// Mitsubishi GX Works2 project: 단속동작   PLC: Q02/Q02H

PROGRAM MAIN
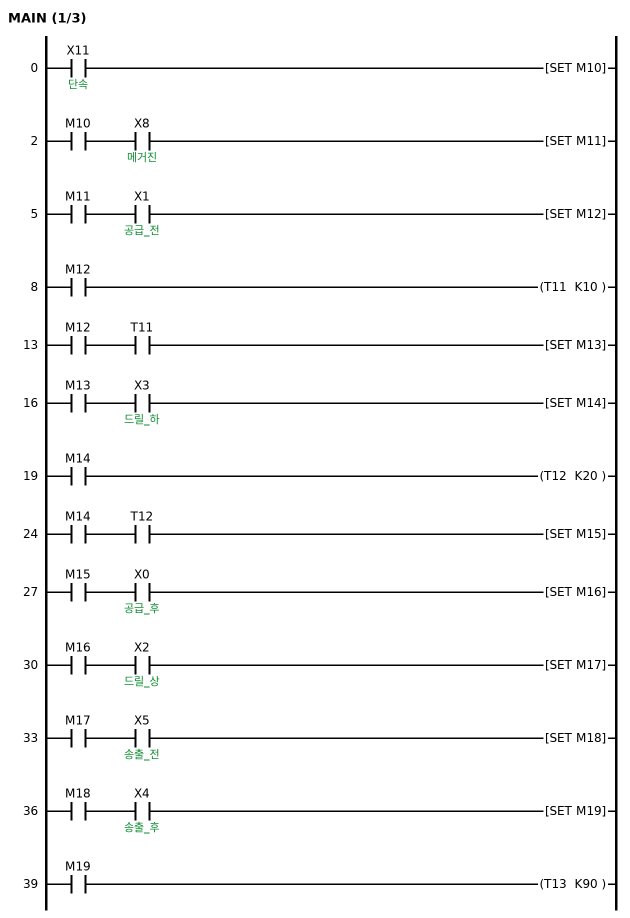
0     LD      X11  ; 단속
      SET     M10
2     LD      M10
      AND     X8  ; 메거진
      SET     M11
5     LD      M11
      AND     X1  ; 공급_전
      SET     M12
8     LD      M12
      OUT     T11 K10
13    LD      M12
      AND     T11
      SET     M13
16    LD      M13
      AND     X3  ; 드릴_하
      SET     M14
19    LD      M14
      OUT     T12 K20
24    LD      M14
      AND     T12
      SET     M15
27    LD      M15
      AND     X0  ; 공급_후
      SET     M16
30    LD      M16
      AND     X2  ; 드릴_상
      SET     M17
33    LD      M17
      AND     X5  ; 송출_전
      SET     M18
36    LD      M18
      AND     X4  ; 송출_후
      SET     M19
39    LD      M19
      OUT     T13 K90
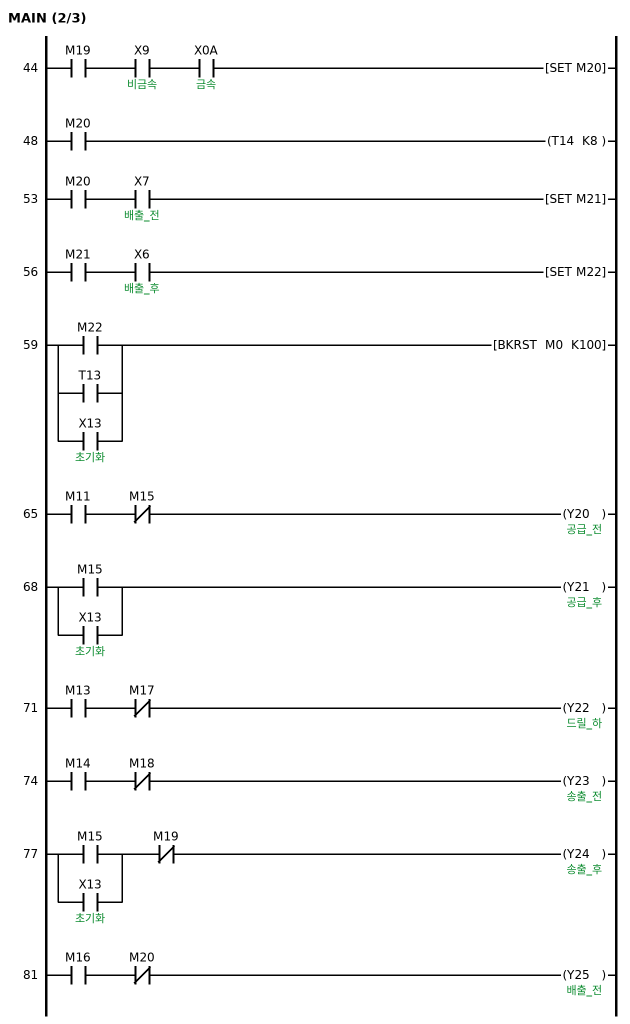
44    LD      M19
      AND     X9  ; 비금속
      AND     X0A  ; 금속
      SET     M20
48    LD      M20
      OUT     T14 K8
53    LD      M20
      AND     X7  ; 배출_전
      SET     M21
56    LD      M21
      AND     X6  ; 배출_후
      SET     M22
59    LD      M22
      OR      T13
      OR      X13  ; 초기화
      BKRST   M0 K100
65    LD      M11
      ANI     M15
      OUT     Y20  ; 공급_전
68    LD      M15
      OR      X13  ; 초기화
      OUT     Y21  ; 공급_후
71    LD      M13
      ANI     M17
      OUT     Y22  ; 드릴_하
74    LD      M14
      ANI     M18
      OUT     Y23  ; 송출_전
77    LD      M15
      OR      X13  ; 초기화
      ANI     M19
      OUT     Y24  ; 송출_후
81    LD      M16
      ANI     M20
      OUT     Y25  ; 배출_전
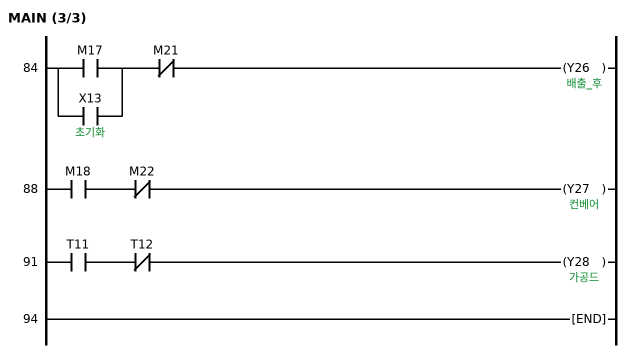
84    LD      M17
      OR      X13  ; 초기화
      ANI     M21
      OUT     Y26  ; 배출_후
88    LD      M18
      ANI     M22
      OUT     Y27  ; 컨베어
91    LD      T11
      ANI     T12
      OUT     Y28  ; 가공드
94    END
END_PROGRAM

// device comments not shown above
X10  ; 테스트
X12  ; 연속
Y29  ; 적색
Y2A  ; 황색
Y2B  ; 녹색
